FUNCTION_BLOCK FB_Assert IMPLEMENTS I_Assert
VAR_INPUT
END_VAR
VAR_OUTPUT
	fbList:					FB_ListSTRING;
	nAssert:				DINT;
	nPassed:				DINT;
	nSkipped:				DINT;
	nFailures:				DINT;
	nErrors:				DINT;
END_VAR
VAR
	fbBuilder:				FB_StringBuilder;
END_VAR

METHOD PUBLIC M_Assert
VAR_INPUT
END_VAR
IF nSkipped = 0 THEN
	nAssert:= nAssert + 1;
END_IF
END_METHOD

METHOD PUBLIC M_Equals_Array_BOOL : I_Assert
VAR_IN_OUT
	Expected:			ARRAY [*] OF BOOL;		// Expected as array of bool
	Actual:				ARRAY [*] OF BOOL;		// Actual as array of bool
END_VAR
VAR_INPUT
	Message:			STRING(255);			// Message as string
END_VAR

VAR
	nIndex:				DINT;
END_VAR
M_Equals_Array_BOOL:= THIS^;
M_Assert();
IF LOWER_BOUND(Expected, 1) <> LOWER_BOUND(Actual, 1) THEN
	M_Failure('', Message);
ELSIF UPPER_BOUND(Expected, 1) <> UPPER_BOUND(Actual, 1) THEN
	M_Failure('', Message);
ELSE
	FOR nIndex:= LOWER_BOUND(Expected, 1) TO UPPER_BOUND(Expected, 1) DO
		IF Expected[nIndex] <> Actual[nIndex] THEN	
			fbBuilder.M_Reset();
			fbBuilder.M_Append('Index = "');
			fbBuilder.M_Append(DINT_TO_STRING(nIndex));
			fbBuilder.M_Append('" Expected = "');
			fbBuilder.M_Append(BOOL_TO_STRING(Expected[nIndex]));
			fbBuilder.M_Append('" Actual = "');
			fbBuilder.M_Append(BOOL_TO_STRING(Actual[nIndex]));
			fbBuilder.M_Append('"');
			M_Failure(fbBuilder.M_ToString(), Message);
			RETURN;
		END_IF
	END_FOR
	M_Passed();
END_IF
END_METHOD

METHOD PUBLIC M_Equals_Array_BYTE : I_Assert
VAR_IN_OUT
	Expected:			ARRAY [*] OF BOOL;	// Expected as array of byte
	Actual:				ARRAY [*] OF BOOL;	// Actual as array of byte
END_VAR                                   
VAR_INPUT                                 
	Message:			STRING(255);     	 // Message as string
END_VAR

VAR
	nIndex:				DINT;
END_VAR
M_Equals_Array_BYTE:= THIS^;
M_Assert();
IF LOWER_BOUND(Expected, 1) <> LOWER_BOUND(Actual, 1) THEN
	M_Failure('', Message);
ELSIF UPPER_BOUND(Expected, 1) <> UPPER_BOUND(Actual, 1) THEN
	M_Failure('', Message);
ELSE
	FOR nIndex:= LOWER_BOUND(Expected, 1) TO UPPER_BOUND(Expected, 1) DO
		IF Expected[nIndex] <> Actual[nIndex] THEN	
			fbBuilder.M_Reset();
			fbBuilder.M_Append('Index = "');
			fbBuilder.M_Append(DINT_TO_STRING(nIndex));
			fbBuilder.M_Append('" Expected = "');
			fbBuilder.M_Append(BOOL_TO_STRING(Expected[nIndex]));
			fbBuilder.M_Append('" Actual = "');
			fbBuilder.M_Append(BOOL_TO_STRING(Actual[nIndex]));
			fbBuilder.M_Append('"');
			M_Failure(fbBuilder.M_ToString(), Message);
			RETURN;
		END_IF
	END_FOR
	M_Passed();
END_IF
END_METHOD

METHOD PUBLIC M_Equals_Array_DINT : I_Assert
VAR_IN_OUT
	Expected:			ARRAY [*] OF DINT;	// Expected as array of dint
	Actual:				ARRAY [*] OF DINT;	// Actual as array of dint
END_VAR                                   
VAR_INPUT                                 
	Message:			STRING(255);       // Message as string
END_VAR

VAR
	nIndex:				DINT;
END_VAR
M_Equals_Array_DINT:= THIS^;
M_Assert();
IF LOWER_BOUND(Expected, 1) <> LOWER_BOUND(Actual, 1) THEN
	M_Failure('', Message);
ELSIF UPPER_BOUND(Expected, 1) <> UPPER_BOUND(Actual, 1) THEN
	M_Failure('', Message);
ELSE
	FOR nIndex:= LOWER_BOUND(Expected, 1) TO UPPER_BOUND(Expected, 1) DO
		IF Expected[nIndex] <> Actual[nIndex] THEN	
			fbBuilder.M_Reset();
			fbBuilder.M_Append('Index = "');
			fbBuilder.M_Append(DINT_TO_STRING(nIndex));
			fbBuilder.M_Append('" Expected = "');
			fbBuilder.M_Append(DINT_TO_STRING(Expected[nIndex]));
			fbBuilder.M_Append('" Actual = "');
			fbBuilder.M_Append(DINT_TO_STRING(Actual[nIndex]));
			fbBuilder.M_Append('"');
			M_Failure(fbBuilder.M_ToString(), Message);
			RETURN;
		END_IF
	END_FOR
	M_Passed();
END_IF
END_METHOD

METHOD PUBLIC M_Equals_Array_INT : I_Assert
VAR_IN_OUT
	Expected:			ARRAY [*] OF INT;	// Expected as array of int
	Actual:				ARRAY [*] OF INT;	// Actual as array of int
END_VAR                                  
VAR_INPUT                                
	Message:			STRING(255);      // Message as string
END_VAR

VAR
	nIndex:				DINT;
END_VAR
M_Equals_Array_INT:= THIS^;
M_Assert();
IF LOWER_BOUND(Expected, 1) <> LOWER_BOUND(Actual, 1) THEN
	M_Failure('', Message);
ELSIF UPPER_BOUND(Expected, 1) <> UPPER_BOUND(Actual, 1) THEN
	M_Failure('', Message);
ELSE
	FOR nIndex:= LOWER_BOUND(Expected, 1) TO UPPER_BOUND(Expected, 1) DO
		IF Expected[nIndex] <> Actual[nIndex] THEN	
			fbBuilder.M_Reset();
			fbBuilder.M_Append('Index = "');
			fbBuilder.M_Append(DINT_TO_STRING(nIndex));
			fbBuilder.M_Append('" Expected = "');
			fbBuilder.M_Append(INT_TO_STRING(Expected[nIndex]));
			fbBuilder.M_Append('" Actual = "');
			fbBuilder.M_Append(INT_TO_STRING(Actual[nIndex]));
			fbBuilder.M_Append('"');
			M_Failure(fbBuilder.M_ToString(), Message);
			RETURN;
		END_IF
	END_FOR
	M_Passed();
END_IF
END_METHOD

METHOD PUBLIC M_Equals_Array_LINT : I_Assert
VAR_IN_OUT
	Expected:			ARRAY [*] OF LINT;	// Expected as array of lint
	Actual:				ARRAY [*] OF LINT;	// Actual as array of lint
END_VAR                                   
VAR_INPUT                                 
	Message:			STRING(255);       // Message as string
END_VAR

VAR
	nIndex:				DINT;
END_VAR
M_Equals_Array_LINT:= THIS^;
M_Assert();
IF LOWER_BOUND(Expected, 1) <> LOWER_BOUND(Actual, 1) THEN
	M_Failure('', Message);
ELSIF UPPER_BOUND(Expected, 1) <> UPPER_BOUND(Actual, 1) THEN
	M_Failure('', Message);
ELSE
	FOR nIndex:= LOWER_BOUND(Expected, 1) TO UPPER_BOUND(Expected, 1) DO
		IF Expected[nIndex] <> Actual[nIndex] THEN	
			fbBuilder.M_Reset();
			fbBuilder.M_Append('Index = "');
			fbBuilder.M_Append(DINT_TO_STRING(nIndex));
			fbBuilder.M_Append('" Expected = "');
			fbBuilder.M_Append(LINT_TO_STRING(Expected[nIndex]));
			fbBuilder.M_Append('" Actual = "');
			fbBuilder.M_Append(LINT_TO_STRING(Actual[nIndex]));
			fbBuilder.M_Append('"');
			M_Failure(fbBuilder.M_ToString(), Message);
			RETURN;
		END_IF
	END_FOR
	M_Passed();
END_IF
END_METHOD

METHOD PUBLIC M_Equals_Array_LREAL : I_Assert
VAR_IN_OUT
	Expected:			ARRAY [*] OF LREAL;	// Expected as array of lreal
	Actual:				ARRAY [*] OF LREAL;	// Actual as array of lreal
END_VAR                                    
VAR_INPUT                                  
	Tolerance:			LREAL;              // Tolerance as lreal
	Message:			STRING(255);		// Message as string
END_VAR

VAR
	nIndex:				DINT;
END_VAR
M_Equals_Array_LREAL:= THIS^;
M_Assert();
IF LOWER_BOUND(Expected, 1) <> LOWER_BOUND(Actual, 1) THEN
	M_Failure('', Message);
ELSIF UPPER_BOUND(Expected, 1) <> UPPER_BOUND(Actual, 1) THEN
	M_Failure('', Message);
ELSE
	FOR nIndex:= LOWER_BOUND(Expected, 1) TO UPPER_BOUND(Expected, 1) DO
		IF ABS(Expected[nIndex] - Actual[nIndex]) > ABS(Tolerance) THEN	
			fbBuilder.M_Reset();
			fbBuilder.M_Append('Index = "');
			fbBuilder.M_Append(DINT_TO_STRING(nIndex));
			fbBuilder.M_Append('" Expected = "');
			fbBuilder.M_Append(LREAL_TO_STRING(Expected[nIndex]));
			fbBuilder.M_Append('" Actual = "');
			fbBuilder.M_Append(LREAL_TO_STRING(Actual[nIndex]));
			fbBuilder.M_Append('"');
			M_Failure(fbBuilder.M_ToString(), Message);
			RETURN;
		END_IF
	END_FOR
	M_Passed();
END_IF
END_METHOD

METHOD PUBLIC M_Equals_Array_REAL : I_Assert
VAR_IN_OUT
	Expected:			ARRAY [*] OF REAL;	// Expected as array of real
	Actual:				ARRAY [*] OF REAL;	// Actual as array of real
END_VAR                                   
VAR_INPUT                                 
	Tolerance:			REAL;             	// Tolerance as real
	Message:			STRING(255);      	// Message as string
END_VAR

VAR
	nIndex:				DINT;
END_VAR
M_Equals_Array_REAL:= THIS^;
M_Assert();
IF LOWER_BOUND(Expected, 1) <> LOWER_BOUND(Actual, 1) THEN
	M_Failure('', Message);
ELSIF UPPER_BOUND(Expected, 1) <> UPPER_BOUND(Actual, 1) THEN
	M_Failure('', Message);
ELSE
	FOR nIndex:= LOWER_BOUND(Expected, 1) TO UPPER_BOUND(Expected, 1) DO
		IF ABS(Expected[nIndex] - Actual[nIndex]) > ABS(Tolerance) THEN	
			fbBuilder.M_Reset();
			fbBuilder.M_Append('Index = "');
			fbBuilder.M_Append(DINT_TO_STRING(nIndex));
			fbBuilder.M_Append('" Expected = "');
			fbBuilder.M_Append(REAL_TO_STRING(Expected[nIndex]));
			fbBuilder.M_Append('" Actual = "');
			fbBuilder.M_Append(REAL_TO_STRING(Actual[nIndex]));
			fbBuilder.M_Append('"');
			M_Failure(fbBuilder.M_ToString(), Message);
			RETURN;
		END_IF
	END_FOR
	M_Passed();
END_IF
END_METHOD

METHOD PUBLIC M_Equals_BOOL : I_Assert
VAR_INPUT
	Expected:			BOOL;				// Expected as bool
    Actual:				BOOL;           	// Actual as bool
	Message:			STRING(255);    	// Message as string
END_VAR
M_Assert();
IF Expected = Actual THEN
	M_Passed();
ELSE
	fbBuilder.M_Reset();
	fbBuilder.M_Append('Expected = "');
	fbBuilder.M_Append(BOOL_TO_STRING(Expected));
	fbBuilder.M_Append('" Actual = "');
	fbBuilder.M_Append(BOOL_TO_STRING(Actual));
	fbBuilder.M_Append('"');
	M_Failure(fbBuilder.M_ToString(), Message);
END_IF
M_Equals_BOOL:= THIS^;
END_METHOD

METHOD PUBLIC M_Equals_BYTE : I_Assert
VAR_INPUT
	Expected:			BYTE;			// Expected as byte
    Actual:				BYTE;           // Actual as byte
	Message:			STRING(255);    // Message as string
END_VAR
M_Assert();
IF Expected = Actual THEN
	M_Passed();
ELSE
	fbBuilder.M_Reset();
	fbBuilder.M_Append('Expected = "');
	fbBuilder.M_Append(BYTE_TO_STRING(Expected));
	fbBuilder.M_Append('" Actual = "');
	fbBuilder.M_Append(BYTE_TO_STRING(Actual));
	fbBuilder.M_Append('"');
	M_Failure(fbBuilder.M_ToString(), Message);
END_IF
M_Equals_BYTE:= THIS^;
END_METHOD

METHOD PUBLIC M_Equals_DINT : I_Assert
VAR_INPUT
	Expected:			DINT;			// Expected as dint
    Actual:				DINT;           // Actual as dint
	Message:			STRING(255);    // Message as string
END_VAR
M_Assert();
IF Expected = Actual THEN
	M_Passed();
ELSE
	fbBuilder.M_Reset();
	fbBuilder.M_Append('Expected = "');
	fbBuilder.M_Append(DINT_TO_STRING(Expected));
	fbBuilder.M_Append('" Actual = "');
	fbBuilder.M_Append(DINT_TO_STRING(Actual));
	fbBuilder.M_Append('"');
	M_Failure(fbBuilder.M_ToString(), Message);
END_IF
M_Equals_DINT:= THIS^;
END_METHOD

METHOD PUBLIC M_Equals_INT : I_Assert
VAR_INPUT
	Expected:			INT;			// Expected as int
    Actual:				INT;            // Actual as int
	Message:			STRING(255);    // Message as string
END_VAR
M_Assert();
IF Expected = Actual THEN
	M_Passed();
ELSE
	fbBuilder.M_Reset();
	fbBuilder.M_Append('Expected = "');
	fbBuilder.M_Append(INT_TO_STRING(Expected));
	fbBuilder.M_Append('" Actual = "');
	fbBuilder.M_Append(INT_TO_STRING(Actual));
	fbBuilder.M_Append('"');
	M_Failure(fbBuilder.M_ToString(), Message);
END_IF
M_Equals_INT:= THIS^;
END_METHOD

METHOD PUBLIC M_Equals_LINT : I_Assert
VAR_INPUT
	Expected:			LINT;			// Expected as lint
    Actual:				LINT;           // Actual as lint
	Message:			STRING(255);    // Message as string
END_VAR
M_Assert();
IF Expected = Actual THEN
	M_Passed();
ELSE
	fbBuilder.M_Reset();
	fbBuilder.M_Append('Expected = "');
	fbBuilder.M_Append(LINT_TO_STRING(Expected));
	fbBuilder.M_Append('" Actual = "');
	fbBuilder.M_Append(LINT_TO_STRING(Actual));
	fbBuilder.M_Append('"');
	M_Failure(fbBuilder.M_ToString(), Message);
END_IF
M_Equals_LINT:= THIS^;
END_METHOD

METHOD PUBLIC M_Equals_LREAL : I_Assert
VAR_INPUT
	Expected:			LREAL;				// Expected as lreal
    Actual:				LREAL;              // Actual as lreal
	Tolerance:			LREAL;             	// Tolerance as lreal         
	Message:			STRING(255);		// Message as string
END_VAR
M_Assert();
IF LrealIsNaN(Expected) THEN
	M_Failure('', Concat('Expected is NaN ', Message));
ELSIF LrealIsNaN(Actual) THEN
	M_Failure('', Concat('Actual is NaN ', Message));	
ELSIF LrealIsNaN(Tolerance) THEN
	M_Failure('', Concat('Tolerance is NaN ', Message));	
ELSIF ABS(Expected - Actual) <= ABS(Tolerance) THEN
	M_Passed();
ELSE
	fbBuilder.M_Reset();
	fbBuilder.M_Append('Expected = "');
	fbBuilder.M_Append(LREAL_TO_STRING(Expected));
	fbBuilder.M_Append('" Actual = "');
	fbBuilder.M_Append(LREAL_TO_STRING(Actual));
	fbBuilder.M_Append('" Tolerance = "');
	fbBuilder.M_Append(LREAL_TO_STRING(Tolerance));
	fbBuilder.M_Append('"');
	M_Failure(fbBuilder.M_ToString(), Message);
END_IF
M_Equals_LREAL:= THIS^;
END_METHOD

METHOD PUBLIC M_Equals_REAL : I_Assert
VAR_INPUT
	Expected:			REAL;			// Expected as real
    Actual:				REAL;           // Actual as real
	Tolerance:			REAL;           // Tolerance as real    
	Message:			STRING(255);    // Message as string
END_VAR
M_Assert();
IF RealIsNaN(Expected) THEN
	M_Failure('', Concat('Expected is NaN ', Message));
ELSIF RealIsNaN(Actual) THEN
	M_Failure('', Concat('Actual is NaN ', Message));	
ELSIF RealIsNaN(Tolerance) THEN
	M_Failure('', Concat('Tolerance is NaN ', Message));	
ELSIF ABS(Expected - Actual) <= ABS(Tolerance) THEN
	M_Passed();
ELSE
	fbBuilder.M_Reset();
	fbBuilder.M_Append('Expected = "');
	fbBuilder.M_Append(LREAL_TO_STRING(Expected));
	fbBuilder.M_Append('" Actual = "');
	fbBuilder.M_Append(LREAL_TO_STRING(Actual));
	fbBuilder.M_Append('" Tolerance = "');
	fbBuilder.M_Append(LREAL_TO_STRING(Tolerance));
	fbBuilder.M_Append('"');
	M_Failure(fbBuilder.M_ToString(), Message);
END_IF
M_Equals_REAL:= THIS^;
END_METHOD

METHOD PUBLIC M_Equals_STRING : I_Assert
VAR_INPUT
	Expected:			STRING(255);		// Expected as string
    Actual:				STRING(255);        // Actual as string
	Message:			STRING(255);      	// Message as string  
END_VAR
M_Assert();
IF Expected = Actual THEN
	M_Passed();
ELSE
	fbBuilder.M_Reset();
	fbBuilder.M_Append('Expected = "');
	fbBuilder.M_Append(Expected);
	fbBuilder.M_Append('" Actual = "');
	fbBuilder.M_Append(Actual);
	fbBuilder.M_Append('"');
	M_Failure(fbBuilder.M_ToString(), Message);
END_IF
M_Equals_STRING:= THIS^;
END_METHOD

METHOD PUBLIC M_Equals_TIME : I_Assert
VAR_INPUT
	Expected:			TIME;				// Expected as time
    Actual:				TIME;               // Actual as time
	Tolerance:			TIME;               // Tolerance as time    
	Message:			STRING(255);        // Message as string
END_VAR
M_Assert();
IF ABS(Expected - Actual) <= ABS(Tolerance) THEN
	M_Passed();
ELSE
	fbBuilder.M_Reset();
	fbBuilder.M_Append('Expected = "');
	fbBuilder.M_Append(TIME_TO_STRING(Expected));
	fbBuilder.M_Append('" Actual = "');
	fbBuilder.M_Append(TIME_TO_STRING(Actual));
	fbBuilder.M_Append('" Tolerance = "');
	fbBuilder.M_Append(TIME_TO_STRING(Tolerance));
	fbBuilder.M_Append('"');
	M_Failure(fbBuilder.M_ToString(), Message);
END_IF
M_Equals_TIME:= THIS^;
END_METHOD

METHOD PUBLIC M_Equals_UDINT : I_Assert
VAR_INPUT
	Expected:			UDINT;			// Expected as udint
    Actual:				UDINT;          // Actual as udint
	Message:			STRING(255);   	// Message as string
END_VAR
M_Assert();
IF Expected = Actual THEN
	M_Passed();
ELSE
	fbBuilder.M_Reset();
	fbBuilder.M_Append('Expected = "');
	fbBuilder.M_Append(UDINT_TO_STRING(Expected));
	fbBuilder.M_Append('" Actual = "');
	fbBuilder.M_Append(UDINT_TO_STRING(Actual));
	fbBuilder.M_Append('"');
	M_Failure(fbBuilder.M_ToString(), Message);
END_IF
M_Equals_UDINT:= THIS^;
END_METHOD

METHOD PUBLIC M_Equals_UINT : I_Assert
VAR_INPUT
	Expected:			UINT;			// Expected as uint
    Actual:				UINT;           // Actual as uint
	Message:			STRING(255);    // Message as string
END_VAR
M_Assert();
IF Expected = Actual THEN
	M_Passed();
ELSE
	fbBuilder.M_Reset();
	fbBuilder.M_Append('Expected = "');
	fbBuilder.M_Append(UINT_TO_STRING(Expected));
	fbBuilder.M_Append('" Actual = "');
	fbBuilder.M_Append(UINT_TO_STRING(Actual));
	fbBuilder.M_Append('"');
	M_Failure(fbBuilder.M_ToString(), Message);
END_IF
M_Equals_UINT:= THIS^;
END_METHOD

METHOD PUBLIC M_Equals_ULINT : I_Assert
VAR_INPUT
	Expected:			ULINT;			// Expected as ulint
    Actual:				ULINT;          // Actual as ulint
	Message:			STRING(255);    // Message as string
END_VAR
M_Assert();
IF Expected = Actual THEN
	M_Passed();
ELSE
	fbBuilder.M_Reset();
	fbBuilder.M_Append('Expected = "');
	fbBuilder.M_Append(ULINT_TO_STRING(Expected));
	fbBuilder.M_Append('" Actual = "');
	fbBuilder.M_Append(ULINT_TO_STRING(Actual));
	fbBuilder.M_Append('"');
	M_Failure(fbBuilder.M_ToString(), Message);
END_IF
M_Equals_ULINT:= THIS^;
END_METHOD

METHOD PUBLIC M_Equals_WSTRING : I_Assert
VAR_INPUT
	Expected:			WSTRING(255);		// Expected as wstring
    Actual:				WSTRING(255);       // Actual as wstring
	Message:			STRING(255);        // Message as string
END_VAR
M_Assert();
IF Expected = Actual THEN
	M_Passed();
ELSE
	fbBuilder.M_Reset();
	fbBuilder.M_Append('Expected = "');
	fbBuilder.M_Append(WSTRING_TO_STRING(Expected));
	fbBuilder.M_Append('" Actual = "');
	fbBuilder.M_Append(WSTRING_TO_STRING(Actual));
	fbBuilder.M_Append('"');
	M_Failure(fbBuilder.M_ToString(), Message);
END_IF
M_Equals_WSTRING:= THIS^;
END_METHOD

METHOD PUBLIC M_Error
VAR_INPUT
	Data:				STRING(255);
	Message:			STRING(255);
END_VAR
IF nSkipped = 0 THEN
	fbBuilder.M_Reset();
	fbBuilder.M_Append('$T$T$T<error message="');
	fbBuilder.M_Append(Message);
	fbBuilder.M_Append('" type="ArithmeticError">');
	fbBuilder.M_Append(Data);	
	fbBuilder.M_Append('"</error>');
	fbList.M_Add(fbBuilder.M_ToString());
	nErrors:= nErrors + 1;
END_IF
END_METHOD

METHOD PUBLIC M_Failure
VAR_INPUT
	Data:				STRING(255);
	Message:			STRING(255);
END_VAR
IF nSkipped = 0 THEN
	fbBuilder.M_Reset();
	fbBuilder.M_Append('$T$T$T<failure message="');
	fbBuilder.M_Append(Message);
	fbBuilder.M_Append('" type="AssertionError">');
	fbBuilder.M_Append(Data);
	fbBuilder.M_Append('"</failure>');
	fbList.M_Add(fbBuilder.M_ToString());
	nFailures:= nFailures + 1;
END_IF
END_METHOD

METHOD PUBLIC M_IsTRUE : I_Assert
VAR_INPUT
    Actual:				BOOL;				// Actual as bool
	Message:			STRING(255);        // Message as string
END_VAR
M_Assert();
IF Actual THEN
	M_Passed();
ELSE
	M_Failure('Actual = FALSE', Message);
	nFailures:= nFailures + 1;
END_IF
M_IsTRUE:= THIS^;
END_METHOD

METHOD PUBLIC M_Passed
VAR_INPUT
END_VAR
IF nSkipped = 0 THEN
	nPassed:= nPassed + 1;
END_IF
END_METHOD

METHOD PUBLIC M_Reset : I_Assert
VAR_INPUT
END_VAR
fbList.M_Clear();
nAssert:= 0;
nPassed:= 0;
nSkipped:= 0;
nFailures:= 0;
nErrors:= 0;
M_Reset:= THIS^;
END_METHOD

METHOD PUBLIC M_Skip
VAR_INPUT
	Message:			STRING(255);	// Message as string
END_VAR
fbList.M_Clear();
nAssert:= 0;
nPassed:= 0;
nFailures:= 0;
nErrors:= 0;
fbBuilder.M_Reset();
fbBuilder.M_Append('$T$T$T<skipped message="');
fbBuilder.M_Append(Message);
fbBuilder.M_Append('" />');
fbList.M_Add(fbBuilder.M_ToString());
nSkipped:= nSkipped + 1;
END_METHOD

METHOD PUBLIC M_TcError : I_Assert
VAR_INPUT
	ErrorId:			UDINT;			// ErrorId as UDINT
	Message:			STRING(255);	// Message as string
END_VAR
VAR
	eError:				E_AdsError:= ErrorId;
END_VAR
M_Assert();
fbBuilder.M_Reset();
IF ErrorId = E_AdsErr.NOERR THEN
	M_Passed();
ELSE
	fbBuilder.M_Reset();
	fbBuilder.M_Append('Expected = "');
	fbBuilder.M_Append(TO_STRING(E_AdsError.NOERR));
	fbBuilder.M_Append('" Actual = "');
	fbBuilder.M_Append(TO_STRING(eError));
	fbBuilder.M_Append('"');
	M_Failure(fbBuilder.M_ToString(), Message);
END_IF
M_TcError:= THIS^;
END_METHOD

END_FUNCTION_BLOCK

(* stored: Version 1.1.0.1
   POU FB_Assert: Id {a8219960-23df-08de-19e5-3265dc5cd828}, SpecialFunc None
   Method M_Assert: Id {20d02a5f-db58-0c6c-14cd-0b5cd69f1cdb}
   Method M_Equals_Array_BOOL: Id {f134011c-e659-0f0f-1451-e11b2d1801b6}
   Method M_Equals_Array_BYTE: Id {12f09544-1af8-0ebe-07a7-8b9c32b9d2dc}
   Method M_Equals_Array_DINT: Id {518ae4ab-060a-09e2-266f-8d59ac7249b8}
   Method M_Equals_Array_INT: Id {6713325b-4c44-0e26-2bb7-5e725aa270d3}
   Method M_Equals_Array_LINT: Id {ad7b55f1-407d-0125-1100-b2f5a1a335ce}
   Method M_Equals_Array_LREAL: Id {c66fd740-f5b0-0aea-32aa-9f9e8cd1f3c8}
   Method M_Equals_Array_REAL: Id {4fd08f76-ba10-092b-0f97-d99ee406f12f}
   Method M_Equals_BOOL: Id {a59ebe08-8964-0b2c-38a4-ac8145e6076b}
   Method M_Equals_BYTE: Id {2d0157fb-a7a4-0a24-2f21-b00692b22401}
   Method M_Equals_DINT: Id {472197bd-33d6-0fc3-0f19-0526022a1a63}
   Method M_Equals_INT: Id {69d1cbc7-70c0-0cef-01a9-39c278d3ddf8}
   Method M_Equals_LINT: Id {a849c410-b14f-0b59-2551-ae0df6d9a14d}
   Method M_Equals_LREAL: Id {56afa40f-43c1-0c87-2e3a-7092c4bb5d6b}
   Method M_Equals_REAL: Id {d6abdbdc-3ed4-0597-3832-aa884ad8510e}
   Method M_Equals_STRING: Id {be4cf22a-d59c-479d-91df-27b8c49cf405}
   Method M_Equals_TIME: Id {91b48555-653d-0553-104e-334d1e902474}
   Method M_Equals_UDINT: Id {dab23cde-89d2-0c20-3b51-ea863cfc23a2}
   Method M_Equals_UINT: Id {d4264b4a-bfbe-0a03-22f6-a7578de8f804}
   Method M_Equals_ULINT: Id {6a3deaae-41c3-057d-0ef8-285e9e3cbbcc}
   Method M_Equals_WSTRING: Id {d57eeb77-552a-03e8-31d9-648afdaf68b1}
   Method M_Error: Id {8fb01682-0d3e-09d1-1052-e80c2a25c45c}
   Method M_Failure: Id {c1dc23cc-f885-0540-1115-b7058773bd0a}
   Method M_IsTRUE: Id {ff21833d-ba1f-05de-0ce2-388ab8c48e28}
   Method M_Passed: Id {0da5074d-f435-0060-10d7-5f55502ee455}
   Method M_Reset: Id {968629c2-18de-07f2-0ab0-109e8e7d42c9}
   Method M_Skip: Id {01e03b07-71f0-0cb8-3278-37acfad51370}
   Method M_TcError: Id {afc6c894-8d15-0f9c-362a-c323312b5010} *)
